// TIA Portal V18 export
FUNCTION "FilmInSafeZoneDeterminator" : Void   // FC18, FBD
{ S7_Optimized_Access := 'TRUE' }
VERSION : 0.1
// stored: AutoNumber true, IsIECCheckEnabled false, SetENOAutomatically false, UDAEnableTagReadback false
   VAR_INPUT
      X : Real;
      x_min : Real;
      x_max : Real;
      Y : Real;
      y_min : Real;
      y_max : Real;
      FILM_MODE : Bool;
      par_dist_arrived : Real;
   END_VAR
   VAR_OUTPUT
      WITHIN_SAFE_ZONE : Bool;
   END_VAR
   VAR_TEMP
      loc_x_safe : Bool;
      loc_y_safe : Bool;
      loc_is_safe : Bool;
      x_min_loc : Real;
      x_max_loc : Real;
      y_min_loc : Real;
      y_max_loc : Real;
      loc_par_dist_arrived : Real;
   END_VAR
BEGIN

REGION Network 2 (SCL)
   #loc_par_dist_arrived := 3 * #par_dist_arrived;

   #x_min_loc := #x_min - #loc_par_dist_arrived;
   #x_max_loc := #x_max + #loc_par_dist_arrived;

   #y_min_loc := #y_min - #loc_par_dist_arrived;
   #y_max_loc := #y_max + #loc_par_dist_arrived;
END_REGION

REGION Network 3
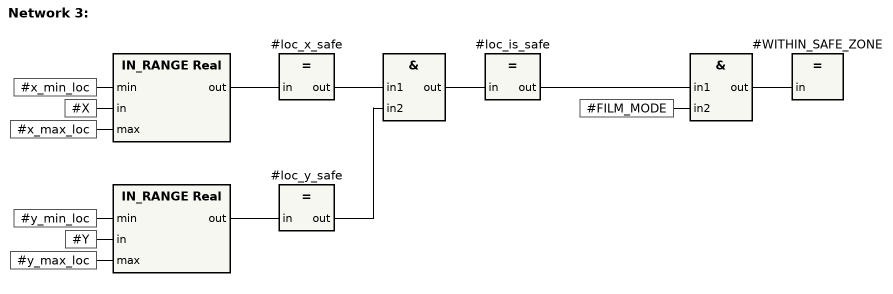
   #loc_x_safe := (#x_min_loc <= #X) AND (#X <= #x_max_loc);
   #loc_y_safe := (#y_min_loc <= #Y) AND (#Y <= #y_max_loc);
   #loc_is_safe := #loc_x_safe AND #loc_y_safe;
   #WITHIN_SAFE_ZONE := #loc_is_safe AND #FILM_MODE;
END_REGION
END_FUNCTION
